DECL PDAT PPDAT515={VEL 100.0,ACC 100.0,APO_DIST 100.0}
DECL E6POS XP770={x 834.883606,y -646.192993,z 1419.58496,a -154.975098,b 4.24509811,c -178.286499,s 2,t 10,e1 0.0,e2 0.0,e3 0.0,e4 0.0,e5 0.0,e6 0.0}
DECL FDAT FP770={TOOL_NO 1,BASE_NO 0,IPO_FRAME #BASE}
DECL PDAT PPDAT516={VEL 100.0,ACC 100.0,APO_DIST 100.0}
DECL E6POS XP771={x 884.407715,y -646.247375,z 1213.34998,a -154.963196,b 4.23633385,c -178.281204,s 2,t 10,e1 0.0,e2 0.0,e3 0.0,e4 0.0,e5 0.0,e6 0.0}
DECL FDAT FP771={TOOL_NO 1,BASE_NO 0,IPO_FRAME #BASE}
DECL PDAT PPDAT517={VEL 100.0,ACC 100.0,APO_DIST 100.0}
DECL E6POS XP772={x 884.420776,y -646.274414,z 1177.65503,a -154.965607,b 4.23612499,c -178.276794,s 2,t 10,e1 0.0,e2 0.0,e3 0.0,e4 0.0,e5 0.0,e6 0.0}
DECL FDAT FP772={TOOL_NO 1,BASE_NO 0,IPO_FRAME #BASE}
DECL LDAT LCPDAT225={VEL 2.0,ACC 100.0,APO_DIST 100.0,APO_FAC 50.0}
DECL E6POS XP773={x 956.251587,y -672.142273,z 1177.66296,a -154.965607,b 4.23677397,c -178.275497,s 2,t 10,e1 0.0,e2 0.0,e3 0.0,e4 0.0,e5 0.0,e6 0.0}
DECL FDAT FP773={TOOL_NO 1,BASE_NO 0,IPO_FRAME #BASE}
DECL LDAT LCPDAT226={VEL 2.0,ACC 100.0,APO_DIST 100.0,APO_FAC 50.0}
DECL E6POS XP774={x 956.253784,y -672.147217,z 1253.29004,a -154.965393,b 4.2372551,c -178.274506,s 2,t 10,e1 0.0,e2 0.0,e3 0.0,e4 0.0,e5 0.0,e6 0.0}
DECL FDAT FP774={TOOL_NO 1,BASE_NO 0,IPO_FRAME #BASE}
DECL LDAT LCPDAT227={VEL 2.0,ACC 100.0,APO_DIST 100.0,APO_FAC 50.0}
DECL E6POS XP775={x 956.25708,y -672.15332,z 1341.07397,a -154.9655,b 4.2373929,c -178.274094,s 2,t 10,e1 0.0,e2 0.0,e3 0.0,e4 0.0,e5 0.0,e6 0.0}
DECL FDAT FP775={TOOL_NO 1,BASE_NO 0,IPO_FRAME #BASE}
DECL PDAT PPDAT518={VEL 100.0,ACC 100.0,APO_DIST 100.0}
DECL E6POS XP776={x 956.26123,y 621.372192,z 1488.15198,a -155.259399,b 5.91821718,c 178.473007,s 2,t 43,e1 0.0,e2 0.0,e3 0.0,e4 0.0,e5 0.0,e6 0.0}
DECL FDAT FP776={TOOL_NO 1,BASE_NO 0,IPO_FRAME #BASE}
DECL PDAT PPDAT519={VEL 100.0,ACC 100.0,APO_DIST 100.0}
DECL E6POS XP777={x 951.221008,y 1494.92102,z 1417.13904,a 164.741592,b -1.48251903,c 173.650696,s 2,t 43,e1 0.0,e2 0.0,e3 0.0,e4 0.0,e5 0.0,e6 0.0}
DECL FDAT FP777={TOOL_NO 1,BASE_NO 0,IPO_FRAME #BASE}
DECL PDAT PPDAT520={VEL 100.0,ACC 100.0,APO_DIST 100.0}
DECL E6POS XP778={x 951.218811,y 1494.91003,z 1304.31799,a 164.741501,b -1.48264694,c 173.651398,s 2,t 43,e1 0.0,e2 0.0,e3 0.0,e4 0.0,e5 0.0,e6 0.0}
DECL FDAT FP778={TOOL_NO 1,BASE_NO 0,IPO_FRAME #BASE}
DECL LDAT LCPDAT228={VEL 2.0,ACC 100.0,APO_DIST 100.0,APO_FAC 50.0}
DECL E6POS XP779={x 951.21698,y 1494.91504,z 1203.42395,a 164.741592,b -1.48277903,c 173.651398,s 2,t 43,e1 0.0,e2 0.0,e3 0.0,e4 0.0,e5 0.0,e6 0.0}
DECL FDAT FP779={TOOL_NO 1,BASE_NO 0,IPO_FRAME #BASE}
DECL LDAT LCPDAT229={VEL 2.0,ACC 100.0,APO_DIST 100.0,APO_FAC 50.0}
DECL E6POS XP780={x 781.836426,y 1615.77795,z 1203.41504,a 164.741699,b -1.48282301,c 173.651199,s 2,t 43,e1 0.0,e2 0.0,e3 0.0,e4 0.0,e5 0.0,e6 0.0}
DECL FDAT FP780={TOOL_NO 1,BASE_NO 0,IPO_FRAME #BASE}
DECL LDAT LCPDAT230={VEL 2.0,ACC 100.0,APO_DIST 100.0,APO_FAC 50.0}
DECL E6POS XP781={x 781.839783,y 1615.78406,z 1295.63196,a 164.741196,b -1.48269701,c 173.650696,s 2,t 43,e1 0.0,e2 0.0,e3 0.0,e4 0.0,e5 0.0,e6 0.0}
DECL FDAT FP781={TOOL_NO 1,BASE_NO 0,IPO_FRAME #BASE}
DECL PDAT PPDAT521={VEL 100.0,ACC 100.0,APO_DIST 100.0}
DECL E6POS XP782={x 781.841492,y 1615.78699,z 1625.56396,a 164.740997,b -1.48261797,c 173.650497,s 2,t 43,e1 0.0,e2 0.0,e3 0.0,e4 0.0,e5 0.0,e6 0.0}
DECL FDAT FP782={TOOL_NO 1,BASE_NO 0,IPO_FRAME #BASE}
DECL PDAT PPDAT522={VEL 100.0,ACC 100.0,APO_DIST 100.0}
DECL E6POS XP783={x 781.886414,y 50.4748688,z 1625.57104,a -152.987396,b 4.59010792,c 178.606796,s 2,t 11,e1 0.0,e2 0.0,e3 0.0,e4 0.0,e5 0.0,e6 0.0}
DECL FDAT FP783={TOOL_NO 1,BASE_NO 0,IPO_FRAME #BASE}
DECL PDAT PPDAT523={VEL 100.0,ACC 100.0,APO_DIST 100.0}
DECL E6POS XP784={x 1625.51196,y 50.4724808,z 1091.81201,a -152.987701,b 4.59131098,c 178.607605,s 2,t 11,e1 0.0,e2 0.0,e3 0.0,e4 0.0,e5 0.0,e6 0.0}
DECL FDAT FP784={TOOL_NO 1,BASE_NO 0,IPO_FRAME #BASE}
DECL PDAT PPDAT524={VEL 100.0,ACC 100.0,APO_DIST 100.0}
DECL E6POS XP785={x 1936.96106,y 50.3517113,z 1091.52197,a 169.965393,b 30.0970707,c 148.691498,s 2,t 10,e1 0.0,e2 0.0,e3 0.0,e4 0.0,e5 0.0,e6 0.0}
DECL FDAT FP785={TOOL_NO 1,BASE_NO 0,IPO_FRAME #BASE}
DECL PDAT PPDAT525={VEL 100.0,ACC 100.0,APO_DIST 100.0}
DECL E6POS XP786={x 2177.73804,y -308.035889,z 1091.83203,a 91.7171021,b 5.48031807,c 146.144806,s 2,t 42,e1 0.0,e2 0.0,e3 0.0,e4 0.0,e5 0.0,e6 0.0}
DECL FDAT FP786={TOOL_NO 1,BASE_NO 0,IPO_FRAME #BASE}
DECL PDAT PPDAT526={VEL 100.0,ACC 100.0,APO_DIST 100.0}
DECL E6POS XP787={x 1894.03699,y -621.732422,z 1187.06897,a 25.7903595,b -5.24155807,c 179.080307,s 2,t 42,e1 0.0,e2 0.0,e3 0.0,e4 0.0,e5 0.0,e6 0.0}
DECL FDAT FP787={TOOL_NO 1,BASE_NO 0,IPO_FRAME #BASE}
DECL PDAT PPDAT527={VEL 100.0,ACC 100.0,APO_DIST 100.0}
DECL E6POS XP788={x 1882.03296,y -621.668518,z 1187.04199,a 25.7881699,b -5.23810196,c 179.0793,s 2,t 42,e1 0.0,e2 0.0,e3 0.0,e4 0.0,e5 0.0,e6 0.0}
DECL FDAT FP788={TOOL_NO 1,BASE_NO 0,IPO_FRAME #BASE}
DECL LDAT LCPDAT231={VEL 2.0,ACC 100.0,APO_DIST 100.0,APO_FAC 50.0}
DECL E6POS XP789={x 1807.823,y -621.600098,z 1187.02002,a 25.1856403,b -5.23544598,c 179.079895,s 2,t 42,e1 0.0,e2 0.0,e3 0.0,e4 0.0,e5 0.0,e6 0.0}
DECL FDAT FP789={TOOL_NO 1,BASE_NO 0,IPO_FRAME #BASE}
DECL LDAT LCPDAT232={VEL 2.0,ACC 100.0,APO_DIST 100.0,APO_FAC 50.0}
DECL E6POS XP790={x 1807.828,y -621.599976,z 1272.56396,a 25.1849709,b -5.2358942,c 179.080093,s 2,t 42,e1 0.0,e2 0.0,e3 0.0,e4 0.0,e5 0.0,e6 0.0}
DECL FDAT FP790={TOOL_NO 1,BASE_NO 0,IPO_FRAME #BASE}
DECL LDAT LCPDAT233={VEL 2.0,ACC 100.0,APO_DIST 100.0,APO_FAC 50.0}
DECL E6POS XP791={x 1807.82104,y -621.602295,z 1311.28894,a 25.1842403,b -5.23504496,c 179.080795,s 2,t 42,e1 0.0,e2 0.0,e3 0.0,e4 0.0,e5 0.0,e6 0.0}
DECL FDAT FP791={TOOL_NO 1,BASE_NO 0,IPO_FRAME #BASE}
DECL PDAT PPDAT528={VEL 100.0,ACC 100.0,APO_DIST 100.0}
DECL E6POS XP792={x 1807.82495,y 498.553192,z 1311.28796,a 25.1833591,b -5.23463488,c 179.080795,s 2,t 35,e1 0.0,e2 0.0,e3 0.0,e4 0.0,e5 0.0,e6 0.0}
DECL FDAT FP792={TOOL_NO 1,BASE_NO 0,IPO_FRAME #BASE}
DECL PDAT PPDAT529={VEL 100.0,ACC 100.0,APO_DIST 100.0}
DECL E6POS XP793={x 1629.39404,y 957.296875,z 1392.64502,a -14.3889599,b -2.57446599,c -174.841293,s 2,t 43,e1 0.0,e2 0.0,e3 0.0,e4 0.0,e5 0.0,e6 0.0}
DECL FDAT FP793={TOOL_NO 1,BASE_NO 0,IPO_FRAME #BASE}
DECL PDAT PPDAT530={VEL 100.0,ACC 100.0,APO_DIST 100.0}
DECL E6POS XP794={x 1629.39099,y 957.29303,z 1270.86804,a -14.3891497,b -2.57352996,c -174.841599,s 2,t 43,e1 0.0,e2 0.0,e3 0.0,e4 0.0,e5 0.0,e6 0.0}
DECL FDAT FP794={TOOL_NO 1,BASE_NO 0,IPO_FRAME #BASE}
DECL PDAT PPDAT531={VEL 100.0,ACC 100.0,APO_DIST 100.0}
DECL E6POS XP795={x 1629.39795,y 957.297913,z 1263.79199,a -14.3884897,b -2.57415891,c -174.840897,s 2,t 43,e1 0.0,e2 0.0,e3 0.0,e4 0.0,e5 0.0,e6 0.0}
DECL FDAT FP795={TOOL_NO 1,BASE_NO 0,IPO_FRAME #BASE}
DECL LDAT LCPDAT234={VEL 2.0,ACC 100.0,APO_DIST 100.0,APO_FAC 50.0}
DECL E6POS XP796={x 1629.39294,y 957.290588,z 1205.66602,a -14.3889904,b -2.573524,c -174.841293,s 2,t 43,e1 0.0,e2 0.0,e3 0.0,e4 0.0,e5 0.0,e6 0.0}
DECL FDAT FP796={TOOL_NO 1,BASE_NO 0,IPO_FRAME #BASE}
DECL LDAT LCPDAT235={VEL 2.0,ACC 100.0,APO_DIST 100.0,APO_FAC 50.0}
DECL E6POS XP797={x 1751.35901,y 834.430481,z 1205.68005,a -14.3898897,b -2.57414389,c -174.840302,s 2,t 43,e1 0.0,e2 0.0,e3 0.0,e4 0.0,e5 0.0,e6 0.0}
DECL FDAT FP797={TOOL_NO 1,BASE_NO 0,IPO_FRAME #BASE}
DECL LDAT LCPDAT236={VEL 2.0,ACC 100.0,APO_DIST 100.0,APO_FAC 50.0}
DECL E6POS XP798={x 1751.36096,y 834.434082,z 1290.125,a -14.39009,b -2.57477689,c -174.840103,s 2,t 43,e1 0.0,e2 0.0,e3 0.0,e4 0.0,e5 0.0,e6 0.0}
DECL FDAT FP798={TOOL_NO 1,BASE_NO 0,IPO_FRAME #BASE}
DECL PDAT PPDAT532={VEL 100.0,ACC 100.0,APO_DIST 100.0}
DECL E6POS XP799={x 1482.72302,y 101.339798,z 1842.39502,a -14.3908005,b -2.57482505,c -174.840393,s 2,t 43,e1 0.0,e2 0.0,e3 0.0,e4 0.0,e5 0.0,e6 0.0}
DECL FDAT FP799={TOOL_NO 1,BASE_NO 0,IPO_FRAME #BASE}
DECL PDAT PPDAT533={VEL 100.0,ACC 100.0,APO_DIST 100.0}
DECL E6POS XP800={x 1967.19495,y -1208.297,z 1007.40997,a 30.6325607,b -2.68640089,c 176.940903,s 2,t 42,e1 0.0,e2 0.0,e3 0.0,e4 0.0,e5 0.0,e6 0.0}
DECL FDAT FP800={TOOL_NO 1,BASE_NO 0,IPO_FRAME #BASE}
DECL PDAT PPDAT534={VEL 100.0,ACC 100.0,APO_DIST 100.0}
DECL E6POS XP801={x 1867.01794,y -1528.33398,z 676.013306,a 26.0535393,b -2.69201303,c 176.927597,s 2,t 42,e1 0.0,e2 0.0,e3 0.0,e4 0.0,e5 0.0,e6 0.0}
DECL FDAT FP801={TOOL_NO 1,BASE_NO 0,IPO_FRAME #BASE}
DECL PDAT PPDAT535={VEL 100.0,ACC 100.0,APO_DIST 100.0}
DECL E6POS XP802={x 1867.14905,y -1528.302,z 632.177185,a 26.0634403,b -2.69869804,c 176.917206,s 2,t 42,e1 0.0,e2 0.0,e3 0.0,e4 0.0,e5 0.0,e6 0.0}
DECL FDAT FP802={TOOL_NO 1,BASE_NO 0,IPO_FRAME #BASE}
DECL LDAT LCPDAT237={VEL 2.0,ACC 100.0,APO_DIST 100.0,APO_FAC 50.0}
DECL E6POS XP803={x 1803.28406,y -1528.18005,z 632.140503,a 26.0650692,b -2.69497204,c 176.921204,s 2,t 42,e1 0.0,e2 0.0,e3 0.0,e4 0.0,e5 0.0,e6 0.0}
DECL FDAT FP803={TOOL_NO 1,BASE_NO 0,IPO_FRAME #BASE}
DECL LDAT LCPDAT238={VEL 2.0,ACC 100.0,APO_DIST 100.0,APO_FAC 50.0}
DECL E6POS XP804={x 1803.28699,y -1528.19104,z 666.373779,a 26.0654392,b -2.69498992,c 176.920303,s 2,t 42,e1 0.0,e2 0.0,e3 0.0,e4 0.0,e5 0.0,e6 0.0}
DECL FDAT FP804={TOOL_NO 1,BASE_NO 0,IPO_FRAME #BASE}
DECL LDAT LCPDAT239={VEL 2.0,ACC 100.0,APO_DIST 100.0,APO_FAC 50.0}
DECL E6POS XP805={x 1803.29004,y -1528.18799,z 707.782471,a 26.0653191,b -2.69489288,c 176.920105,s 2,t 42,e1 0.0,e2 0.0,e3 0.0,e4 0.0,e5 0.0,e6 0.0}
DECL FDAT FP805={TOOL_NO 1,BASE_NO 0,IPO_FRAME #BASE}
DECL PDAT PPDAT536={VEL 100.0,ACC 100.0,APO_DIST 100.0}
DECL E6POS XP806={x 1849.71899,y 504.765503,z 982.790527,a 25.7066708,b -3.66189194,c -178.073196,s 2,t 43,e1 0.0,e2 0.0,e3 0.0,e4 0.0,e5 0.0,e6 0.0}
DECL FDAT FP806={TOOL_NO 1,BASE_NO 0,IPO_FRAME #BASE}
DECL PDAT PPDAT537={VEL 100.0,ACC 100.0,APO_DIST 100.0}
DECL E6POS XP807={x 1526.51599,y 887.347717,z 1356.229,a 119.449997,b -0.79832828,c 176.833496,s 2,t 43,e1 0.0,e2 0.0,e3 0.0,e4 0.0,e5 0.0,e6 0.0}
DECL FDAT FP807={TOOL_NO 1,BASE_NO 0,IPO_FRAME #BASE}
DECL PDAT PPDAT538={VEL 100.0,ACC 100.0,APO_DIST 100.0}
DECL E6POS XP808={x 1117.29504,y 985.80957,z 1503.50098,a -103.3563,b 6.37956905,c -178.578705,s 2,t 11,e1 0.0,e2 0.0,e3 0.0,e4 0.0,e5 0.0,e6 0.0}
DECL FDAT FP808={TOOL_NO 1,BASE_NO 0,IPO_FRAME #BASE}
DECL PDAT PPDAT539={VEL 100.0,ACC 100.0,APO_DIST 100.0}
DECL E6POS XP809={x 1110.35498,y 986.373596,z 1199.61401,a -104.191902,b 6.3782239,c -178.580399,s 2,t 11,e1 0.0,e2 0.0,e3 0.0,e4 0.0,e5 0.0,e6 0.0}
DECL FDAT FP809={TOOL_NO 1,BASE_NO 0,IPO_FRAME #BASE}
DECL LDAT LCPDAT240={VEL 2.0,ACC 100.0,APO_DIST 100.0,APO_FAC 50.0}
DECL E6POS XP810={x 1110.35706,y 986.37439,z 1177.31006,a -104.191597,b 6.37824202,c -178.580093,s 2,t 11,e1 0.0,e2 0.0,e3 0.0,e4 0.0,e5 0.0,e6 0.0}
DECL FDAT FP810={TOOL_NO 1,BASE_NO 0,IPO_FRAME #BASE}
DECL LDAT LCPDAT241={VEL 2.0,ACC 100.0,APO_DIST 100.0,APO_FAC 50.0}
DECL E6POS XP811={x 1060.698,y 922.256287,z 1177.30701,a -104.191704,b 6.3783679,c -178.580093,s 2,t 11,e1 0.0,e2 0.0,e3 0.0,e4 0.0,e5 0.0,e6 0.0}
DECL FDAT FP811={TOOL_NO 1,BASE_NO 0,IPO_FRAME #BASE}
DECL LDAT LCPDAT242={VEL 2.0,ACC 100.0,APO_DIST 100.0,APO_FAC 50.0}
DECL E6POS XP812={x 1060.70605,y 922.260193,z 1248.45898,a -104.1922,b 6.37897682,c -178.580002,s 2,t 11,e1 0.0,e2 0.0,e3 0.0,e4 0.0,e5 0.0,e6 0.0}
DECL FDAT FP812={TOOL_NO 1,BASE_NO 0,IPO_FRAME #BASE}
DECL LDAT LCPDAT243={VEL 2.0,ACC 100.0,APO_DIST 100.0,APO_FAC 50.0}
DECL E6POS XP813={x 1060.70801,y 922.260986,z 1325.92102,a -104.193199,b 6.37862921,c -178.5802,s 2,t 11,e1 0.0,e2 0.0,e3 0.0,e4 0.0,e5 0.0,e6 0.0}
DECL FDAT FP813={TOOL_NO 1,BASE_NO 0,IPO_FRAME #BASE}
DECL PDAT PPDAT540={VEL 100.0,ACC 100.0,APO_DIST 100.0}
DECL E6POS XP814={x 1007.14001,y -531.034973,z 1325.93103,a -154.515793,b 6.37904882,c -178.579803,s 2,t 10,e1 0.0,e2 0.0,e3 0.0,e4 0.0,e5 0.0,e6 0.0}
DECL FDAT FP814={TOOL_NO 1,BASE_NO 0,IPO_FRAME #BASE}
DECL PDAT PPDAT541={VEL 100.0,ACC 100.0,APO_DIST 100.0}
DECL E6POS XP815={x 662.151917,y -1577.61401,z 1042.82104,a -155.219803,b 2.91244411,c -175.284103,s 2,t 10,e1 0.0,e2 0.0,e3 0.0,e4 0.0,e5 0.0,e6 0.0}
DECL FDAT FP815={TOOL_NO 1,BASE_NO 0,IPO_FRAME #BASE}
DECL PDAT PPDAT542={VEL 100.0,ACC 100.0,APO_DIST 100.0}
DECL E6POS XP816={x 595.804382,y -1577.60999,z 610.217285,a -155.219498,b 2.91238999,c -175.284607,s 2,t 10,e1 0.0,e2 0.0,e3 0.0,e4 0.0,e5 0.0,e6 0.0}
DECL FDAT FP816={TOOL_NO 1,BASE_NO 0,IPO_FRAME #BASE}
DECL PDAT PPDAT543={VEL 100.0,ACC 100.0,APO_DIST 100.0}
DECL E6POS XP817={x 677.520874,y -1577.67395,z 616.163086,a -155.236404,b 0.510486484,c -174.949493,s 2,t 10,e1 0.0,e2 0.0,e3 0.0,e4 0.0,e5 0.0,e6 0.0}
DECL FDAT FP817={TOOL_NO 1,BASE_NO 0,IPO_FRAME #BASE}
DECL PDAT PPDAT544={VEL 100.0,ACC 100.0,APO_DIST 100.0}
DECL E6POS XP818={x 680.30188,y -1577.672,z 616.161621,a -155.236694,b 0.510483205,c -174.949905,s 2,t 10,e1 0.0,e2 0.0,e3 0.0,e4 0.0,e5 0.0,e6 0.0}
DECL FDAT FP818={TOOL_NO 1,BASE_NO 0,IPO_FRAME #BASE}
DECL LDAT LCPDAT244={VEL 2.0,ACC 100.0,APO_DIST 100.0,APO_FAC 50.0}
DECL E6POS XP819={x 729.268921,y -1577.66602,z 614.958984,a -155.235901,b 0.510274529,c -174.950394,s 2,t 10,e1 0.0,e2 0.0,e3 0.0,e4 0.0,e5 0.0,e6 0.0}
DECL FDAT FP819={TOOL_NO 1,BASE_NO 0,IPO_FRAME #BASE}
DECL LDAT LCPDAT245={VEL 2.0,ACC 100.0,APO_DIST 100.0,APO_FAC 50.0}
DECL E6POS XP820={x 729.266174,y -1577.66895,z 665.128723,a -155.235794,b 0.510224879,c -174.950699,s 2,t 10,e1 0.0,e2 0.0,e3 0.0,e4 0.0,e5 0.0,e6 0.0}
DECL FDAT FP820={TOOL_NO 1,BASE_NO 0,IPO_FRAME #BASE}
DECL LDAT LCPDAT246={VEL 2.0,ACC 100.0,APO_DIST 100.0,APO_FAC 50.0}
DECL E6POS XP821={x 729.262085,y -1577.66003,z 715.29657,a -155.235703,b 0.510212183,c -174.951202,s 2,t 10,e1 0.0,e2 0.0,e3 0.0,e4 0.0,e5 0.0,e6 0.0}
DECL FDAT FP821={TOOL_NO 1,BASE_NO 0,IPO_FRAME #BASE}
DECL PDAT PPDAT545={VEL 100.0,ACC 100.0,APO_DIST 100.0}
DECL E6POS XP822={x 1350.92798,y -438.835693,z 1277.92603,a -155.235504,b 0.510017395,c -174.951096,s 2,t 2,e1 0.0,e2 0.0,e3 0.0,e4 0.0,e5 0.0,e6 0.0}
DECL FDAT FP822={TOOL_NO 1,BASE_NO 0,IPO_FRAME #BASE}
DECL PDAT PPDAT546={VEL 100.0,ACC 100.0,APO_DIST 100.0}
DECL E6POS XP823={x 1350.94495,y -65.3104172,z 1277.97803,a -155.459106,b 3.8784039,c -179.287598,s 2,t 10,e1 0.0,e2 0.0,e3 0.0,e4 0.0,e5 0.0,e6 0.0}
DECL FDAT FP823={TOOL_NO 1,BASE_NO 0,IPO_FRAME #BASE}
DECL PDAT PPDAT547={VEL 100.0,ACC 100.0,APO_DIST 100.0}
DECL E6POS XP824={x 1350.95801,y 508.329315,z 1277.97095,a -103.423302,b 3.87848401,c -179.288406,s 2,t 11,e1 0.0,e2 0.0,e3 0.0,e4 0.0,e5 0.0,e6 0.0}
DECL FDAT FP824={TOOL_NO 1,BASE_NO 0,IPO_FRAME #BASE}
DECL PDAT PPDAT548={VEL 100.0,ACC 100.0,APO_DIST 100.0}
DECL E6POS XP825={x 976.178101,y 799.219421,z 1277.97095,a -103.422897,b 3.87840891,c -179.288498,s 2,t 11,e1 0.0,e2 0.0,e3 0.0,e4 0.0,e5 0.0,e6 0.0}
DECL FDAT FP825={TOOL_NO 1,BASE_NO 0,IPO_FRAME #BASE}
DECL PDAT PPDAT549={VEL 100.0,ACC 100.0,APO_DIST 100.0}
DECL E6POS XP826={x 976.189697,y 799.22113,z 1265.927,a -103.4245,b 3.87825489,c -179.287796,s 2,t 11,e1 0.0,e2 0.0,e3 0.0,e4 0.0,e5 0.0,e6 0.0}
DECL FDAT FP826={TOOL_NO 1,BASE_NO 0,IPO_FRAME #BASE}
DECL LDAT LCPDAT247={VEL 2.0,ACC 100.0,APO_DIST 100.0,APO_FAC 50.0}
DECL E6POS XP827={x 973.25177,y 802.428528,z 1180.17896,a -104.262299,b 3.87858891,c -179.288193,s 2,t 11,e1 0.0,e2 0.0,e3 0.0,e4 0.0,e5 0.0,e6 0.0}
DECL FDAT FP827={TOOL_NO 1,BASE_NO 0,IPO_FRAME #BASE}
DECL LDAT LCPDAT248={VEL 2.0,ACC 100.0,APO_DIST 100.0,APO_FAC 50.0}
DECL E6POS XP828={x 903.986694,y 734.74292,z 1180.17896,a -104.262199,b 3.87883902,c -179.288101,s 2,t 11,e1 0.0,e2 0.0,e3 0.0,e4 0.0,e5 0.0,e6 0.0}
DECL FDAT FP828={TOOL_NO 1,BASE_NO 0,IPO_FRAME #BASE}
DECL LDAT LCPDAT249={VEL 2.0,ACC 100.0,APO_DIST 100.0,APO_FAC 50.0}
DECL E6POS XP829={x 903.989075,y 691.025574,z 1431.854,a -104.2621,b 3.87912607,c -179.287994,s 2,t 11,e1 0.0,e2 0.0,e3 0.0,e4 0.0,e5 0.0,e6 0.0}
DECL FDAT FP829={TOOL_NO 1,BASE_NO 0,IPO_FRAME #BASE}
DECL PDAT PPDAT550={VEL 100.0,ACC 100.0,APO_DIST 100.0}
DECL E6POS XP830={x 1242.453,y 383.157196,z 1431.854,a -65.0922165,b 1.82727897,c -174.843307,s 2,t 11,e1 0.0,e2 0.0,e3 0.0,e4 0.0,e5 0.0,e6 0.0}
DECL FDAT FP830={TOOL_NO 1,BASE_NO 0,IPO_FRAME #BASE}
DECL PDAT PPDAT551={VEL 100.0,ACC 100.0,APO_DIST 100.0}
DECL E6POS XP831={x 1242.526,y -1715.71497,z 1090.12195,a -65.0943909,b 1.824404,c -174.841507,s 2,t 10,e1 0.0,e2 0.0,e3 0.0,e4 0.0,e5 0.0,e6 0.0}
DECL FDAT FP831={TOOL_NO 1,BASE_NO 0,IPO_FRAME #BASE}
DECL PDAT PPDAT552={VEL 100.0,ACC 100.0,APO_DIST 100.0}
DECL E6POS XP832={x 1267.51099,y -2121.16797,z 696.45282,a -64.79319,b -2.43663502,c -176.824097,s 2,t 10,e1 0.0,e2 0.0,e3 0.0,e4 0.0,e5 0.0,e6 0.0}
DECL FDAT FP832={TOOL_NO 1,BASE_NO 0,IPO_FRAME #BASE}
DECL PDAT PPDAT553={VEL 100.0,ACC 100.0,APO_DIST 100.0}
DECL E6POS XP833={x 1268.06104,y -2138.6001,z 629.002625,a -64.8109665,b -2.74127197,c -176.339798,s 2,t 10,e1 0.0,e2 0.0,e3 0.0,e4 0.0,e5 0.0,e6 0.0}
DECL FDAT FP833={TOOL_NO 1,BASE_NO 0,IPO_FRAME #BASE}
DECL LDAT LCPDAT250={VEL 2.0,ACC 100.0,APO_DIST 100.0,APO_FAC 50.0}
DECL E6POS XP834={x 1267.37195,y -2113.87012,z 626.005981,a -64.8136368,b -2.71599889,c -176.349594,s 2,t 10,e1 0.0,e2 0.0,e3 0.0,e4 0.0,e5 0.0,e6 0.0}
DECL FDAT FP834={TOOL_NO 1,BASE_NO 0,IPO_FRAME #BASE}
DECL LDAT LCPDAT251={VEL 2.0,ACC 100.0,APO_DIST 100.0,APO_FAC 50.0}
DECL E6POS XP835={x 1267.10999,y -2080.51807,z 625.848328,a -64.8051834,b -2.70687294,c -176.356506,s 2,t 10,e1 0.0,e2 0.0,e3 0.0,e4 0.0,e5 0.0,e6 0.0}
DECL FDAT FP835={TOOL_NO 1,BASE_NO 0,IPO_FRAME #BASE}
DECL LDAT LCPDAT252={VEL 2.0,ACC 100.0,APO_DIST 100.0,APO_FAC 50.0}
DECL E6POS XP836={x 1267.10901,y -2080.51611,z 624.96228,a -64.8052521,b -2.70639491,c -176.356598,s 2,t 10,e1 0.0,e2 0.0,e3 0.0,e4 0.0,e5 0.0,e6 0.0}
DECL FDAT FP836={TOOL_NO 1,BASE_NO 0,IPO_FRAME #BASE}
DECL LDAT LCPDAT253={VEL 2.0,ACC 100.0,APO_DIST 100.0,APO_FAC 50.0}
DECL E6POS XP837={x 1284.23096,y -2080.74902,z 625.221313,a -64.8089066,b -2.72878504,c -176.344299,s 2,t 10,e1 0.0,e2 0.0,e3 0.0,e4 0.0,e5 0.0,e6 0.0}
DECL FDAT FP837={TOOL_NO 1,BASE_NO 0,IPO_FRAME #BASE}
DECL LDAT LCPDAT254={VEL 2.0,ACC 100.0,APO_DIST 100.0,APO_FAC 50.0}
DECL E6POS XP838={x 1284.21899,y -2080.75,z 674.30957,a -64.8095093,b -2.728158,c -176.344498,s 2,t 10,e1 0.0,e2 0.0,e3 0.0,e4 0.0,e5 0.0,e6 0.0}
DECL FDAT FP838={TOOL_NO 1,BASE_NO 0,IPO_FRAME #BASE}
DECL LDAT LCPDAT255={VEL 2.0,ACC 100.0,APO_DIST 100.0,APO_FAC 50.0}
DECL E6POS XP839={x 1284.21301,y -2080.75098,z 781.889709,a -64.8102188,b -2.72803593,c -176.344498,s 2,t 10,e1 0.0,e2 0.0,e3 0.0,e4 0.0,e5 0.0,e6 0.0}
DECL FDAT FP839={TOOL_NO 1,BASE_NO 0,IPO_FRAME #BASE}
DECL PDAT PPDAT554={VEL 100.0,ACC 100.0,APO_DIST 100.0}
DECL E6POS XP840={x 1284.33301,y 158.871704,z 1306.61304,a -64.8253937,b 1.14583802,c -174.523804,s 2,t 11,e1 0.0,e2 0.0,e3 0.0,e4 0.0,e5 0.0,e6 0.0}
DECL FDAT FP840={TOOL_NO 1,BASE_NO 0,IPO_FRAME #BASE}
DECL PDAT PPDAT555={VEL 100.0,ACC 100.0,APO_DIST 100.0}
DECL E6POS XP841={x 1590.53296,y 626.546387,z 1306.651,a -14.1000004,b -1.28675902,c -174.4617,s 2,t 11,e1 0.0,e2 0.0,e3 0.0,e4 0.0,e5 0.0,e6 0.0}
DECL FDAT FP841={TOOL_NO 1,BASE_NO 0,IPO_FRAME #BASE}
DECL PDAT PPDAT556={VEL 100.0,ACC 100.0,APO_DIST 100.0}
DECL E6POS XP842={x 1716.79199,y 897.809082,z 1262.11096,a -13.9702301,b -1.29123998,c -174.459503,s 2,t 11,e1 0.0,e2 0.0,e3 0.0,e4 0.0,e5 0.0,e6 0.0}
DECL FDAT FP842={TOOL_NO 1,BASE_NO 0,IPO_FRAME #BASE}
DECL PDAT PPDAT557={VEL 100.0,ACC 100.0,APO_DIST 100.0}
DECL E6POS XP843={x 1716.79199,y 897.806274,z 1247.396,a -13.9698601,b -1.29120898,c -174.459,s 2,t 11,e1 0.0,e2 0.0,e3 0.0,e4 0.0,e5 0.0,e6 0.0}
DECL FDAT FP843={TOOL_NO 1,BASE_NO 0,IPO_FRAME #BASE}
DECL LDAT LCPDAT256={VEL 2.0,ACC 100.0,APO_DIST 100.0,APO_FAC 50.0}
DECL E6POS XP844={x 1716.78198,y 897.80249,z 1198.69897,a -13.9701004,b -1.29035699,c -174.459396,s 2,t 11,e1 0.0,e2 0.0,e3 0.0,e4 0.0,e5 0.0,e6 0.0}
DECL FDAT FP844={TOOL_NO 1,BASE_NO 0,IPO_FRAME #BASE}
DECL LDAT LCPDAT257={VEL 2.0,ACC 100.0,APO_DIST 100.0,APO_FAC 50.0}
DECL E6POS XP845={x 1802.52795,y 828.709717,z 1198.69604,a -13.9702501,b -1.29001105,c -174.459305,s 2,t 11,e1 0.0,e2 0.0,e3 0.0,e4 0.0,e5 0.0,e6 0.0}
DECL FDAT FP845={TOOL_NO 1,BASE_NO 0,IPO_FRAME #BASE}
DECL LDAT LCPDAT258={VEL 2.0,ACC 100.0,APO_DIST 100.0,APO_FAC 50.0}
DECL E6POS XP846={x 1802.51294,y 761.127502,z 1198.72302,a -13.9681501,b -1.29168904,c -174.458298,s 2,t 11,e1 0.0,e2 0.0,e3 0.0,e4 0.0,e5 0.0,e6 0.0}
DECL FDAT FP846={TOOL_NO 1,BASE_NO 0,IPO_FRAME #BASE}
DECL PDAT PPDAT558={VEL 100.0,ACC 100.0,APO_DIST 100.0}
DECL E6POS XP847={x 1802.50598,y -336.506287,z 1185.67297,a 118.019897,b 4.52842808,c 174.709198,s 2,t 34,e1 0.0,e2 0.0,e3 0.0,e4 0.0,e5 0.0,e6 0.0}
DECL FDAT FP847={TOOL_NO 1,BASE_NO 0,IPO_FRAME #BASE}
DECL PDAT PPDAT559={VEL 100.0,ACC 100.0,APO_DIST 100.0}
DECL E6POS XP848={x 1270.18604,y -947.062622,z 660.983521,a 112.980698,b 4.33244419,c 178.080505,s 2,t 34,e1 0.0,e2 0.0,e3 0.0,e4 0.0,e5 0.0,e6 0.0}
DECL FDAT FP848={TOOL_NO 1,BASE_NO 0,IPO_FRAME #BASE}
DECL PDAT PPDAT560={VEL 100.0,ACC 100.0,APO_DIST 100.0}
DECL E6POS XP849={x 1286.21497,y -986.133179,z 597.794983,a 112.979897,b 4.33160305,c 178.080902,s 2,t 34,e1 0.0,e2 0.0,e3 0.0,e4 0.0,e5 0.0,e6 0.0}
DECL FDAT FP849={TOOL_NO 1,BASE_NO 0,IPO_FRAME #BASE}
DECL LDAT LCPDAT259={VEL 2.0,ACC 100.0,APO_DIST 100.0,APO_FAC 50.0}
DECL E6POS XP850={x 1286.00305,y -1018.45898,z 597.88147,a 113.2043,b 4.06272316,c 178.724106,s 2,t 34,e1 0.0,e2 0.0,e3 0.0,e4 0.0,e5 0.0,e6 0.0}
DECL FDAT FP850={TOOL_NO 1,BASE_NO 0,IPO_FRAME #BASE}
DECL LDAT LCPDAT260={VEL 2.0,ACC 100.0,APO_DIST 100.0,APO_FAC 50.0}
DECL E6POS XP851={x 1274.45605,y -1018.44501,z 598.83728,a 113.204597,b 4.06176376,c 178.724594,s 2,t 34,e1 0.0,e2 0.0,e3 0.0,e4 0.0,e5 0.0,e6 0.0}
DECL FDAT FP851={TOOL_NO 1,BASE_NO 0,IPO_FRAME #BASE}
DECL LDAT LCPDAT261={VEL 2.0,ACC 100.0,APO_DIST 100.0,APO_FAC 50.0}
DECL E6POS XP852={x 1274.45996,y -1018.448,z 627.330078,a 113.205299,b 4.06202507,c 178.724503,s 2,t 34,e1 0.0,e2 0.0,e3 0.0,e4 0.0,e5 0.0,e6 0.0}
DECL FDAT FP852={TOOL_NO 1,BASE_NO 0,IPO_FRAME #BASE}
DECL LDAT LCPDAT262={VEL 2.0,ACC 100.0,APO_DIST 100.0,APO_FAC 50.0}
DECL E6POS XP853={x 1274.47095,y -1018.46503,z 647.700317,a 113.2052,b 4.06336021,c 178.723801,s 2,t 34,e1 0.0,e2 0.0,e3 0.0,e4 0.0,e5 0.0,e6 0.0}
DECL FDAT FP853={TOOL_NO 1,BASE_NO 0,IPO_FRAME #BASE}
DECL PDAT PPDAT561={VEL 100.0,ACC 100.0,APO_DIST 100.0}
DECL E6POS XP854={x 1274.40405,y 438.174194,z 1449.75903,a 113.028397,b 1.96038795,c 176.1409,s 2,t 35,e1 0.0,e2 0.0,e3 0.0,e4 0.0,e5 0.0,e6 0.0}
DECL FDAT FP854={TOOL_NO 1,BASE_NO 0,IPO_FRAME #BASE}
DECL PDAT PPDAT562={VEL 100.0,ACC 100.0,APO_DIST 100.0}
DECL E6POS XP855={x 1274.41199,y 579.304382,z 1449.76697,a -174.676498,b 7.10730505,c 176.619904,s 2,t 43,e1 0.0,e2 0.0,e3 0.0,e4 0.0,e5 0.0,e6 0.0}
DECL FDAT FP855={TOOL_NO 1,BASE_NO 0,IPO_FRAME #BASE}
DECL PDAT PPDAT563={VEL 100.0,ACC 100.0,APO_DIST 100.0}
DECL E6POS XP856={x 1274.41699,y 964.305115,z 1449.76404,a -153.690308,b 6.61543608,c -179.989594,s 2,t 35,e1 0.0,e2 0.0,e3 0.0,e4 0.0,e5 0.0,e6 0.0}
DECL FDAT FP856={TOOL_NO 1,BASE_NO 0,IPO_FRAME #BASE}
DECL PDAT PPDAT564={VEL 100.0,ACC 100.0,APO_DIST 100.0}
DECL E6POS XP857={x 758.336426,y 1284.67102,z 1449.76001,a 165.206497,b 2.00212693,c 176.736298,s 2,t 35,e1 0.0,e2 0.0,e3 0.0,e4 0.0,e5 0.0,e6 0.0}
DECL FDAT FP857={TOOL_NO 1,BASE_NO 0,IPO_FRAME #BASE}
DECL PDAT PPDAT565={VEL 100.0,ACC 100.0,APO_DIST 100.0}
DECL E6POS XP858={x 865.113892,y 1552.07104,z 1237.68701,a 166.427094,b 2.00283194,c 176.733902,s 2,t 35,e1 0.0,e2 0.0,e3 0.0,e4 0.0,e5 0.0,e6 0.0}
DECL FDAT FP858={TOOL_NO 1,BASE_NO 0,IPO_FRAME #BASE}
DECL PDAT PPDAT566={VEL 100.0,ACC 100.0,APO_DIST 100.0}
DECL E6POS XP859={x 865.110718,y 1552.06494,z 1225.62695,a 166.426804,b 2.00282502,c 176.7341,s 2,t 35,e1 0.0,e2 0.0,e3 0.0,e4 0.0,e5 0.0,e6 0.0}
DECL FDAT FP859={TOOL_NO 1,BASE_NO 0,IPO_FRAME #BASE}
DECL LDAT LCPDAT263={VEL 2.0,ACC 100.0,APO_DIST 100.0,APO_FAC 50.0}
DECL E6POS XP860={x 865.113098,y 1552.06201,z 1174.51501,a 166.426193,b 2.00270891,c 176.733994,s 2,t 35,e1 0.0,e2 0.0,e3 0.0,e4 0.0,e5 0.0,e6 0.0}
DECL FDAT FP860={TOOL_NO 1,BASE_NO 0,IPO_FRAME #BASE}
DECL LDAT LCPDAT264={VEL 2.0,ACC 100.0,APO_DIST 100.0,APO_FAC 50.0}
DECL E6POS XP861={x 739.028076,y 1608.69604,z 1174.51501,a 166.426193,b 2.00264096,c 176.733994,s 2,t 35,e1 0.0,e2 0.0,e3 0.0,e4 0.0,e5 0.0,e6 0.0}
DECL FDAT FP861={TOOL_NO 1,BASE_NO 0,IPO_FRAME #BASE}
DECL LDAT LCPDAT265={VEL 2.0,ACC 100.0,APO_DIST 100.0,APO_FAC 50.0}
DECL E6POS XP862={x 739.030212,y 1608.69299,z 1249.495,a 166.425995,b 2.0026021,c 176.733093,s 2,t 35,e1 0.0,e2 0.0,e3 0.0,e4 0.0,e5 0.0,e6 0.0}
DECL FDAT FP862={TOOL_NO 1,BASE_NO 0,IPO_FRAME #BASE}
DECL PDAT PPDAT567={VEL 100.0,ACC 100.0,APO_DIST 100.0}
DECL E6POS XP863={x 977.82428,y 601.907227,z 1521.28406,a -150.784698,b 2.0027411,c 176.732895,s 2,t 11,e1 0.0,e2 0.0,e3 0.0,e4 0.0,e5 0.0,e6 0.0}
DECL FDAT FP863={TOOL_NO 1,BASE_NO 0,IPO_FRAME #BASE}
DECL PDAT PPDAT568={VEL 100.0,ACC 100.0,APO_DIST 100.0}
DECL E6POS XP864={x 977.828918,y -339.057892,z 1521.28296,a -150.784805,b 2.0027051,c 176.733093,s 2,t 10,e1 0.0,e2 0.0,e3 0.0,e4 0.0,e5 0.0,e6 0.0}
DECL FDAT FP864={TOOL_NO 1,BASE_NO 0,IPO_FRAME #BASE}
DECL PDAT PPDAT569={VEL 100.0,ACC 100.0,APO_DIST 100.0}
DECL E6POS XP865={x 667.386719,y -1536.68201,z 1024.74194,a -155.497299,b 5.11866999,c -174.992004,s 2,t 10,e1 0.0,e2 0.0,e3 0.0,e4 0.0,e5 0.0,e6 0.0}
DECL FDAT FP865={TOOL_NO 1,BASE_NO 0,IPO_FRAME #BASE}
DECL PDAT PPDAT570={VEL 100.0,ACC 100.0,APO_DIST 100.0}
DECL E6POS XP866={x 622.895874,y -1574.84204,z 545.977112,a -155.458801,b 2.811517,c -174.407898,s 2,t 10,e1 0.0,e2 0.0,e3 0.0,e4 0.0,e5 0.0,e6 0.0}
DECL FDAT FP866={TOOL_NO 1,BASE_NO 0,IPO_FRAME #BASE}
DECL PDAT PPDAT571={VEL 100.0,ACC 100.0,APO_DIST 100.0}
DECL E6POS XP867={x 672.657288,y -1574.83606,z 545.976685,a -155.459,b 2.81164193,c -174.408707,s 2,t 10,e1 0.0,e2 0.0,e3 0.0,e4 0.0,e5 0.0,e6 0.0}
DECL FDAT FP867={TOOL_NO 1,BASE_NO 0,IPO_FRAME #BASE}
DECL LDAT LCPDAT266={VEL 2.0,ACC 100.0,APO_DIST 100.0,APO_FAC 50.0}
DECL E6POS XP868={x 721.0354,y -1574.83899,z 545.978271,a -155.458801,b 2.8112781,c -174.408005,s 2,t 10,e1 0.0,e2 0.0,e3 0.0,e4 0.0,e5 0.0,e6 0.0}
DECL FDAT FP868={TOOL_NO 1,BASE_NO 0,IPO_FRAME #BASE}
DECL LDAT LCPDAT267={VEL 2.0,ACC 100.0,APO_DIST 100.0,APO_FAC 50.0}
DECL E6POS XP869={x 724.281128,y -1574.85596,z 573.222107,a -155.458694,b 2.81117201,c -174.406998,s 2,t 10,e1 0.0,e2 0.0,e3 0.0,e4 0.0,e5 0.0,e6 0.0}
DECL FDAT FP869={TOOL_NO 1,BASE_NO 0,IPO_FRAME #BASE}
DECL LDAT LCPDAT268={VEL 2.0,ACC 100.0,APO_DIST 100.0,APO_FAC 50.0}
DECL E6POS XP870={x 724.284973,y -1574.86401,z 633.002014,a -155.458694,b 2.81121707,c -174.406693,s 2,t 10,e1 0.0,e2 0.0,e3 0.0,e4 0.0,e5 0.0,e6 0.0}
DECL FDAT FP870={TOOL_NO 1,BASE_NO 0,IPO_FRAME #BASE}
DECL LDAT LCPDAT269={VEL 2.0,ACC 100.0,APO_DIST 100.0,APO_FAC 50.0}
DECL E6POS XP871={x 724.276611,y -1574.85303,z 730.688904,a -155.460098,b 2.81144595,c -174.407898,s 2,t 10,e1 0.0,e2 0.0,e3 0.0,e4 0.0,e5 0.0,e6 0.0}
DECL FDAT FP871={TOOL_NO 1,BASE_NO 0,IPO_FRAME #BASE}
DECL PDAT PPDAT572={VEL 100.0,ACC 100.0,APO_DIST 100.0}
DECL E6POS XP872={x 1196.31104,y -12.7953701,z 1384.39001,a -155.803299,b 5.08000183,c -179.398697,s 2,t 10,e1 0.0,e2 0.0,e3 0.0,e4 0.0,e5 0.0,e6 0.0}
DECL FDAT FP872={TOOL_NO 1,BASE_NO 0,IPO_FRAME #BASE}
DECL PDAT PPDAT573={VEL 100.0,ACC 100.0,APO_DIST 100.0}
DECL E6POS XP873={x 988.161072,y 807.089172,z 1384.35095,a -104.207802,b 7.43646288,c -177.310806,s 2,t 11,e1 0.0,e2 0.0,e3 0.0,e4 0.0,e5 0.0,e6 0.0}
DECL FDAT FP873={TOOL_NO 1,BASE_NO 0,IPO_FRAME #BASE}
DECL PDAT PPDAT574={VEL 100.0,ACC 100.0,APO_DIST 100.0}
DECL E6POS XP874={x 966.663086,y 799.905518,z 1213.52795,a -104.207497,b 7.43645382,c -177.310394,s 2,t 11,e1 0.0,e2 0.0,e3 0.0,e4 0.0,e5 0.0,e6 0.0}
DECL FDAT FP874={TOOL_NO 1,BASE_NO 0,IPO_FRAME #BASE}
DECL PDAT PPDAT575={VEL 100.0,ACC 100.0,APO_DIST 100.0}
DECL E6POS XP875={x 968.942078,y 800.869324,z 1193.94604,a -104.704903,b 7.43691778,c -177.309402,s 2,t 11,e1 0.0,e2 0.0,e3 0.0,e4 0.0,e5 0.0,e6 0.0}
DECL FDAT FP875={TOOL_NO 1,BASE_NO 0,IPO_FRAME #BASE}
DECL LDAT LCPDAT270={VEL 2.0,ACC 100.0,APO_DIST 100.0,APO_FAC 50.0}
DECL E6POS XP876={x 968.950012,y 800.86908,z 1184.78003,a -104.703697,b 7.43699217,c -177.3078,s 2,t 11,e1 0.0,e2 0.0,e3 0.0,e4 0.0,e5 0.0,e6 0.0}
DECL FDAT FP876={TOOL_NO 1,BASE_NO 0,IPO_FRAME #BASE}
DECL LDAT LCPDAT271={VEL 2.0,ACC 100.0,APO_DIST 100.0,APO_FAC 50.0}
DECL E6POS XP877={x 910.592285,y 742.152527,z 1184.78796,a -104.703499,b 7.43762779,c -177.307297,s 2,t 11,e1 0.0,e2 0.0,e3 0.0,e4 0.0,e5 0.0,e6 0.0}
DECL FDAT FP877={TOOL_NO 1,BASE_NO 0,IPO_FRAME #BASE}
DECL LDAT LCPDAT272={VEL 2.0,ACC 100.0,APO_DIST 100.0,APO_FAC 50.0}
DECL E6POS XP878={x 910.58429,y 742.146606,z 1226.82104,a -104.703697,b 7.43728113,c -177.3078,s 2,t 11,e1 0.0,e2 0.0,e3 0.0,e4 0.0,e5 0.0,e6 0.0}
DECL FDAT FP878={TOOL_NO 1,BASE_NO 0,IPO_FRAME #BASE}
DECL PDAT PPDAT576={VEL 100.0,ACC 100.0,APO_DIST 100.0}
DECL E6POS XP879={x 941.989319,y 683.767883,z 1368.15906,a -104.703598,b 7.43723583,c -177.3078,s 2,t 11,e1 0.0,e2 0.0,e3 0.0,e4 0.0,e5 0.0,e6 0.0}
DECL FDAT FP879={TOOL_NO 1,BASE_NO 0,IPO_FRAME #BASE}
DECL PDAT PPDAT577={VEL 100.0,ACC 100.0,APO_DIST 100.0}
DECL E6POS XP880={x 1528.52197,y 420.196503,z 1368.17505,a 25.5136395,b -4.00302076,c -174.884094,s 2,t 43,e1 0.0,e2 0.0,e3 0.0,e4 0.0,e5 0.0,e6 0.0}
DECL FDAT FP880={TOOL_NO 1,BASE_NO 0,IPO_FRAME #BASE}
DECL PDAT PPDAT578={VEL 100.0,ACC 100.0,APO_DIST 100.0}
DECL E6POS XP881={x 1860.85901,y -1558.21399,z 642.981689,a 25.7883205,b -1.25623298,c 176.261795,s 2,t 34,e1 0.0,e2 0.0,e3 0.0,e4 0.0,e5 0.0,e6 0.0}
DECL FDAT FP881={TOOL_NO 1,BASE_NO 0,IPO_FRAME #BASE}
DECL PDAT PPDAT579={VEL 100.0,ACC 100.0,APO_DIST 100.0}
DECL E6POS XP882={x 1860.66699,y -1529.20898,z 642.863098,a 25.7857208,b -1.25422895,c 176.274002,s 2,t 34,e1 0.0,e2 0.0,e3 0.0,e4 0.0,e5 0.0,e6 0.0}
DECL FDAT FP882={TOOL_NO 1,BASE_NO 0,IPO_FRAME #BASE}
DECL PDAT PPDAT580={VEL 100.0,ACC 100.0,APO_DIST 100.0}
DECL E6POS XP883={x 1838.44995,y -1527.78796,z 608.491882,a 25.75494,b -1.242275,c 176.294006,s 2,t 34,e1 0.0,e2 0.0,e3 0.0,e4 0.0,e5 0.0,e6 0.0}
DECL FDAT FP883={TOOL_NO 1,BASE_NO 0,IPO_FRAME #BASE}
DECL LDAT LCPDAT273={VEL 2.0,ACC 100.0,APO_DIST 100.0,APO_FAC 50.0}
DECL E6POS XP884={x 1799.22998,y -1526.58801,z 608.364685,a 25.7351704,b -1.22906005,c 176.322693,s 2,t 34,e1 0.0,e2 0.0,e3 0.0,e4 0.0,e5 0.0,e6 0.0}
DECL FDAT FP884={TOOL_NO 1,BASE_NO 0,IPO_FRAME #BASE}
DECL LDAT LCPDAT274={VEL 2.0,ACC 100.0,APO_DIST 100.0,APO_FAC 50.0}
DECL E6POS XP885={x 1799.23096,y -1526.59497,z 655.081116,a 25.7347908,b -1.22934604,c 176.322205,s 2,t 34,e1 0.0,e2 0.0,e3 0.0,e4 0.0,e5 0.0,e6 0.0}
DECL FDAT FP885={TOOL_NO 1,BASE_NO 0,IPO_FRAME #BASE}
DECL LDAT LCPDAT275={VEL 2.0,ACC 100.0,APO_DIST 100.0,APO_FAC 50.0}
DECL E6POS XP886={x 1799.22803,y -1526.58496,z 719.989685,a 25.7348709,b -1.22912896,c 176.323105,s 2,t 34,e1 0.0,e2 0.0,e3 0.0,e4 0.0,e5 0.0,e6 0.0}
DECL FDAT FP886={TOOL_NO 1,BASE_NO 0,IPO_FRAME #BASE}
DECL PDAT PPDAT581={VEL 100.0,ACC 100.0,APO_DIST 100.0}
DECL E6POS XP887={x 1799.29004,y -82.3157806,z 720.017517,a 25.6821003,b -2.48299694,c 177.8004,s 2,t 34,e1 0.0,e2 0.0,e3 0.0,e4 0.0,e5 0.0,e6 0.0}
DECL FDAT FP887={TOOL_NO 1,BASE_NO 0,IPO_FRAME #BASE}
DECL PDAT PPDAT582={VEL 100.0,ACC 100.0,APO_DIST 100.0}
DECL E6POS XP888={x 1799.30701,y 860.608582,z 1382.677,a 81.5148468,b -2.00226498,c 175.8414,s 2,t 35,e1 0.0,e2 0.0,e3 0.0,e4 0.0,e5 0.0,e6 0.0}
DECL FDAT FP888={TOOL_NO 1,BASE_NO 0,IPO_FRAME #BASE}
DECL PDAT PPDAT583={VEL 100.0,ACC 100.0,APO_DIST 100.0}
DECL E6POS XP889={x 1609.86401,y 1631.90002,z 1256.89099,a 76.4038315,b -2.0085659,c 175.839798,s 2,t 35,e1 0.0,e2 0.0,e3 0.0,e4 0.0,e5 0.0,e6 0.0}
DECL FDAT FP889={TOOL_NO 1,BASE_NO 0,IPO_FRAME #BASE}
DECL PDAT PPDAT584={VEL 100.0,ACC 100.0,APO_DIST 100.0}
DECL E6POS XP890={x 1609.75696,y 1632.01196,z 1241.46594,a 76.1206207,b -2.85729408,c -178.738403,s 2,t 43,e1 0.0,e2 0.0,e3 0.0,e4 0.0,e5 0.0,e6 0.0}
DECL FDAT FP890={TOOL_NO 1,BASE_NO 0,IPO_FRAME #BASE}
DECL LDAT LCPDAT276={VEL 2.0,ACC 100.0,APO_DIST 100.0,APO_FAC 50.0}
DECL E6POS XP891={x 1609.76404,y 1634.53406,z 1227.97498,a 76.3281784,b -2.85829806,c -178.7397,s 2,t 43,e1 0.0,e2 0.0,e3 0.0,e4 0.0,e5 0.0,e6 0.0}
DECL FDAT FP891={TOOL_NO 1,BASE_NO 0,IPO_FRAME #BASE}
DECL LDAT LCPDAT277={VEL 2.0,ACC 100.0,APO_DIST 100.0,APO_FAC 50.0}
DECL E6POS XP892={x 1609.75696,y 1634.53296,z 1221.46997,a 76.3280411,b -2.85753608,c -178.739502,s 2,t 43,e1 0.0,e2 0.0,e3 0.0,e4 0.0,e5 0.0,e6 0.0}
DECL FDAT FP892={TOOL_NO 1,BASE_NO 0,IPO_FRAME #BASE}
DECL LDAT LCPDAT278={VEL 2.0,ACC 100.0,APO_DIST 100.0,APO_FAC 50.0}
DECL E6POS XP893={x 1660.14001,y 1684.52405,z 1221.47302,a 76.3276825,b -2.858459,c -178.740097,s 2,t 43,e1 0.0,e2 0.0,e3 0.0,e4 0.0,e5 0.0,e6 0.0}
DECL FDAT FP893={TOOL_NO 1,BASE_NO 0,IPO_FRAME #BASE}
DECL LDAT LCPDAT279={VEL 2.0,ACC 100.0,APO_DIST 100.0,APO_FAC 50.0}
DECL E6POS XP894={x 1660.13794,y 1684.521,z 1299.00696,a 76.3268127,b -2.858325,c -178.740097,s 2,t 43,e1 0.0,e2 0.0,e3 0.0,e4 0.0,e5 0.0,e6 0.0}
DECL FDAT FP894={TOOL_NO 1,BASE_NO 0,IPO_FRAME #BASE}
DECL PDAT PPDAT585={VEL 100.0,ACC 100.0,APO_DIST 100.0}
DECL E6POS XP895={x 1660.13794,y 1684.52197,z 1374.20496,a 76.3268738,b -2.85910106,c -178.740601,s 2,t 43,e1 0.0,e2 0.0,e3 0.0,e4 0.0,e5 0.0,e6 0.0}
DECL FDAT FP895={TOOL_NO 1,BASE_NO 0,IPO_FRAME #BASE}
DECL PDAT PPDAT586={VEL 100.0,ACC 100.0,APO_DIST 100.0}
DECL E6POS XP896={x 1675.53296,y 1393.375,z 1577.74597,a 76.3267517,b -2.85850406,c -178.740494,s 2,t 43,e1 0.0,e2 0.0,e3 0.0,e4 0.0,e5 0.0,e6 0.0}
DECL FDAT FP896={TOOL_NO 1,BASE_NO 0,IPO_FRAME #BASE}
DECL PDAT PPDAT587={VEL 100.0,ACC 100.0,APO_DIST 100.0}
DECL E6POS XP897={x 1341.71399,y -974.840027,z 988.560608,a 76.3263092,b -2.85842299,c -178.740997,s 2,t 42,e1 0.0,e2 0.0,e3 0.0,e4 0.0,e5 0.0,e6 0.0}
DECL FDAT FP897={TOOL_NO 1,BASE_NO 0,IPO_FRAME #BASE}
DECL PDAT PPDAT588={VEL 100.0,ACC 100.0,APO_DIST 100.0}
DECL E6POS XP898={x 1248.776,y -913.338989,z 845.195679,a 117.022499,b 1.62681997,c 178.727005,s 2,t 42,e1 0.0,e2 0.0,e3 0.0,e4 0.0,e5 0.0,e6 0.0}
DECL FDAT FP898={TOOL_NO 1,BASE_NO 0,IPO_FRAME #BASE}
DECL PDAT PPDAT589={VEL 100.0,ACC 100.0,APO_DIST 100.0}
DECL E6POS XP899={x 1253.00696,y -913.317383,z 598.303894,a 114.828201,b 1.62474203,c 178.729004,s 2,t 42,e1 0.0,e2 0.0,e3 0.0,e4 0.0,e5 0.0,e6 0.0}
DECL FDAT FP899={TOOL_NO 1,BASE_NO 0,IPO_FRAME #BASE}
DECL PDAT PPDAT590={VEL 100.0,ACC 100.0,APO_DIST 100.0}
DECL E6POS XP900={x 1253.01001,y -978.737122,z 592.641174,a 114.827599,b 1.62485695,c 178.728897,s 2,t 42,e1 0.0,e2 0.0,e3 0.0,e4 0.0,e5 0.0,e6 0.0}
DECL FDAT FP900={TOOL_NO 1,BASE_NO 0,IPO_FRAME #BASE}
DECL LDAT LCPDAT280={VEL 2.0,ACC 100.0,APO_DIST 100.0,APO_FAC 50.0}
DECL E6POS XP901={x 1252.77002,y -1020.51501,z 592.645874,a 114.8349,b 1.82319403,c 179.311798,s 2,t 34,e1 0.0,e2 0.0,e3 0.0,e4 0.0,e5 0.0,e6 0.0}
DECL FDAT FP901={TOOL_NO 1,BASE_NO 0,IPO_FRAME #BASE}
DECL LDAT LCPDAT281={VEL 2.0,ACC 100.0,APO_DIST 100.0,APO_FAC 50.0}
DECL E6POS XP902={x 1263.38403,y -1020.33502,z 594.706116,a 114.819801,b 2.10123897,c 178.699997,s 2,t 42,e1 0.0,e2 0.0,e3 0.0,e4 0.0,e5 0.0,e6 0.0}
DECL FDAT FP902={TOOL_NO 1,BASE_NO 0,IPO_FRAME #BASE}
DECL LDAT LCPDAT282={VEL 2.0,ACC 100.0,APO_DIST 100.0,APO_FAC 50.0}
DECL E6POS XP903={x 1263.38403,y -1020.33502,z 625.024597,a 114.819801,b 2.101403,c 178.699905,s 2,t 42,e1 0.0,e2 0.0,e3 0.0,e4 0.0,e5 0.0,e6 0.0}
DECL FDAT FP903={TOOL_NO 1,BASE_NO 0,IPO_FRAME #BASE}
DECL LDAT LCPDAT283={VEL 2.0,ACC 100.0,APO_DIST 100.0,APO_FAC 50.0}
DECL E6POS XP904={x 1263.38,y -1020.33197,z 688.816284,a 114.819298,b 2.10045004,c 178.700302,s 2,t 42,e1 0.0,e2 0.0,e3 0.0,e4 0.0,e5 0.0,e6 0.0}
DECL FDAT FP904={TOOL_NO 1,BASE_NO 0,IPO_FRAME #BASE}
DECL PDAT PPDAT591={VEL 100.0,ACC 100.0,APO_DIST 100.0}
DECL E6POS XP905={x 1263.38098,y 535.155823,z 1453.13501,a 114.819603,b 2.10045791,c 178.700195,s 2,t 35,e1 0.0,e2 0.0,e3 0.0,e4 0.0,e5 0.0,e6 0.0}
DECL FDAT FP905={TOOL_NO 1,BASE_NO 0,IPO_FRAME #BASE}
DECL PDAT PPDAT592={VEL 100.0,ACC 100.0,APO_DIST 100.0}
DECL E6POS XP906={x 897.335876,y 1571.90503,z 1453.13403,a 164.976303,b 2.10037708,c 178.700394,s 2,t 35,e1 0.0,e2 0.0,e3 0.0,e4 0.0,e5 0.0,e6 0.0}
DECL FDAT FP906={TOOL_NO 1,BASE_NO 0,IPO_FRAME #BASE}
DECL PDAT PPDAT593={VEL 100.0,ACC 100.0,APO_DIST 100.0}
DECL E6POS XP907={x 865.246094,y 1550.27197,z 1230.71497,a 166.390503,b 2.10056996,c 178.699402,s 2,t 35,e1 0.0,e2 0.0,e3 0.0,e4 0.0,e5 0.0,e6 0.0}
DECL FDAT FP907={TOOL_NO 1,BASE_NO 0,IPO_FRAME #BASE}
DECL PDAT PPDAT594={VEL 100.0,ACC 100.0,APO_DIST 100.0}
DECL E6POS XP908={x 865.25177,y 1552.198,z 1212.11304,a 166.391205,b 2.10028696,c 178.698898,s 2,t 35,e1 0.0,e2 0.0,e3 0.0,e4 0.0,e5 0.0,e6 0.0}
DECL FDAT FP908={TOOL_NO 1,BASE_NO 0,IPO_FRAME #BASE}
DECL LDAT LCPDAT284={VEL 2.0,ACC 100.0,APO_DIST 100.0,APO_FAC 50.0}
DECL E6POS XP909={x 866.094482,y 1555.01196,z 1231.22205,a 166.395401,b -0.139191896,c 176.842407,s 2,t 43,e1 0.0,e2 0.0,e3 0.0,e4 0.0,e5 0.0,e6 0.0}
DECL FDAT FP909={TOOL_NO 1,BASE_NO 0,IPO_FRAME #BASE}
DECL LDAT LCPDAT285={VEL 2.0,ACC 100.0,APO_DIST 100.0,APO_FAC 50.0}
DECL E6POS XP910={x 866.09137,y 1555.00598,z 1222.16199,a 166.395294,b -0.139310107,c 176.842804,s 2,t 43,e1 0.0,e2 0.0,e3 0.0,e4 0.0,e5 0.0,e6 0.0}
DECL FDAT FP910={TOOL_NO 1,BASE_NO 0,IPO_FRAME #BASE}
DECL LDAT LCPDAT286={VEL 2.0,ACC 100.0,APO_DIST 100.0,APO_FAC 50.0}
DECL E6POS XP911={x 809.880615,y 1554.99304,z 1222.15698,a 166.394897,b -0.139069393,c 176.843399,s 2,t 43,e1 0.0,e2 0.0,e3 0.0,e4 0.0,e5 0.0,e6 0.0}
DECL FDAT FP911={TOOL_NO 1,BASE_NO 0,IPO_FRAME #BASE}
DECL LDAT LCPDAT287={VEL 2.0,ACC 100.0,APO_DIST 100.0,APO_FAC 50.0}
DECL E6POS XP912={x 699.510376,y 1554.98901,z 1222.15002,a 166.394897,b -0.139277503,c 176.843704,s 2,t 43,e1 0.0,e2 0.0,e3 0.0,e4 0.0,e5 0.0,e6 0.0}
DECL FDAT FP912={TOOL_NO 1,BASE_NO 0,IPO_FRAME #BASE}
DECL PDAT PPDAT595={VEL 100.0,ACC 100.0,APO_DIST 100.0}
DECL E6POS XP913={x 699.511902,y 1554.98499,z 1488.83105,a 166.394501,b -0.139487296,c 176.844101,s 2,t 43,e1 0.0,e2 0.0,e3 0.0,e4 0.0,e5 0.0,e6 0.0}
DECL FDAT FP913={TOOL_NO 1,BASE_NO 0,IPO_FRAME #BASE}
DECL PDAT PPDAT596={VEL 100.0,ACC 100.0,APO_DIST 100.0}
DECL E6POS XP914={x 699.508789,y 538.287781,z 1488.85706,a 166.396896,b -0.138524607,c 176.842697,s 2,t 43,e1 0.0,e2 0.0,e3 0.0,e4 0.0,e5 0.0,e6 0.0}
DECL FDAT FP914={TOOL_NO 1,BASE_NO 0,IPO_FRAME #BASE}
DECL PDAT PPDAT597={VEL 100.0,ACC 100.0,APO_DIST 100.0}
DECL E6POS XP915={x 699.515991,y -1863.35803,z 1488.84802,a -179.705093,b -0.138834104,c 176.842194,s 2,t 10,e1 0.0,e2 0.0,e3 0.0,e4 0.0,e5 0.0,e6 0.0}
DECL FDAT FP915={TOOL_NO 1,BASE_NO 0,IPO_FRAME #BASE}
DECL PDAT PPDAT598={VEL 100.0,ACC 100.0,APO_DIST 100.0}
DECL E6POS XP916={x 1107.23206,y -2206.31201,z 732.711182,a -64.4342194,b -0.146776795,c 176.841003,s 2,t 2,e1 0.0,e2 0.0,e3 0.0,e4 0.0,e5 0.0,e6 0.0}
DECL FDAT FP916={TOOL_NO 1,BASE_NO 0,IPO_FRAME #BASE}
DECL PDAT PPDAT599={VEL 100.0,ACC 100.0,APO_DIST 100.0}
DECL E6POS XP917={x 1277.12903,y -2126.3269,z 663.030579,a -64.4268265,b -0.130556002,c 176.844498,s 2,t 2,e1 0.0,e2 0.0,e3 0.0,e4 0.0,e5 0.0,e6 0.0}
DECL FDAT FP917={TOOL_NO 1,BASE_NO 0,IPO_FRAME #BASE}
DECL PDAT PPDAT600={VEL 100.0,ACC 100.0,APO_DIST 100.0}
DECL E6POS XP918={x 1277.21802,y -2126.26196,z 611.331421,a -64.6608429,b -3.56653905,c -175.942093,s 2,t 10,e1 0.0,e2 0.0,e3 0.0,e4 0.0,e5 0.0,e6 0.0}
DECL FDAT FP918={TOOL_NO 1,BASE_NO 0,IPO_FRAME #BASE}
DECL PDAT PPDAT601={VEL 100.0,ACC 100.0,APO_DIST 100.0}
DECL E6POS XP919={x 1276.80005,y -2112.41504,z 611.11322,a -64.6627884,b -3.54889011,c -175.948807,s 2,t 10,e1 0.0,e2 0.0,e3 0.0,e4 0.0,e5 0.0,e6 0.0}
DECL FDAT FP919={TOOL_NO 1,BASE_NO 0,IPO_FRAME #BASE}
DECL LDAT LCPDAT288={VEL 2.0,ACC 100.0,APO_DIST 100.0,APO_FAC 50.0}
DECL E6POS XP920={x 1276.58801,y -2080.27588,z 611.015381,a -64.6592026,b -3.53906202,c -175.953995,s 2,t 10,e1 0.0,e2 0.0,e3 0.0,e4 0.0,e5 0.0,e6 0.0}
DECL FDAT FP920={TOOL_NO 1,BASE_NO 0,IPO_FRAME #BASE}
DECL LDAT LCPDAT289={VEL 2.0,ACC 100.0,APO_DIST 100.0,APO_FAC 50.0}
DECL E6POS XP921={x 1276.58801,y -2080.28003,z 671.877808,a -64.6594162,b -3.53952503,c -175.954407,s 2,t 10,e1 0.0,e2 0.0,e3 0.0,e4 0.0,e5 0.0,e6 0.0}
DECL FDAT FP921={TOOL_NO 1,BASE_NO 0,IPO_FRAME #BASE}
DECL LDAT LCPDAT290={VEL 2.0,ACC 100.0,APO_DIST 100.0,APO_FAC 50.0}
DECL E6POS XP922={x 1276.58704,y -2080.28296,z 777.328674,a -64.6594772,b -3.53981996,c -175.954697,s 2,t 10,e1 0.0,e2 0.0,e3 0.0,e4 0.0,e5 0.0,e6 0.0}
DECL FDAT FP922={TOOL_NO 1,BASE_NO 0,IPO_FRAME #BASE}
DECL PDAT PPDAT602={VEL 100.0,ACC 100.0,APO_DIST 100.0}
DECL E6POS XP923={x 1276.58801,y -2080.28394,z 1232.85303,a -64.6595078,b -3.54048896,c -175.954605,s 2,t 10,e1 0.0,e2 0.0,e3 0.0,e4 0.0,e5 0.0,e6 0.0}
DECL FDAT FP923={TOOL_NO 1,BASE_NO 0,IPO_FRAME #BASE}
DECL PDAT PPDAT603={VEL 100.0,ACC 100.0,APO_DIST 100.0}
DECL E6POS XP924={x 1276.58606,y 455.985413,z 1340.87097,a -64.7281418,b 1.18211102,c -173.376801,s 2,t 11,e1 0.0,e2 0.0,e3 0.0,e4 0.0,e5 0.0,e6 0.0}
DECL FDAT FP924={TOOL_NO 1,BASE_NO 0,IPO_FRAME #BASE}
DECL PDAT PPDAT604={VEL 100.0,ACC 100.0,APO_DIST 100.0}
DECL E6POS XP925={x 1740.078,y 702.766418,z 1340.85303,a -4.79579878,b 1.18323004,c -173.377304,s 2,t 11,e1 0.0,e2 0.0,e3 0.0,e4 0.0,e5 0.0,e6 0.0}
DECL FDAT FP925={TOOL_NO 1,BASE_NO 0,IPO_FRAME #BASE}
DECL PDAT PPDAT605={VEL 100.0,ACC 100.0,APO_DIST 100.0}
DECL E6POS XP926={x 1710.87805,y 890.413818,z 1240.81897,a -13.7459402,b -1.86556697,c -172.673004,s 2,t 11,e1 0.0,e2 0.0,e3 0.0,e4 0.0,e5 0.0,e6 0.0}
DECL FDAT FP926={TOOL_NO 1,BASE_NO 0,IPO_FRAME #BASE}
DECL LDAT LCPDAT291={VEL 2.0,ACC 100.0,APO_DIST 100.0,APO_FAC 50.0}
DECL E6POS XP927={x 1710.86304,y 892.215027,z 1241.10303,a -13.7396097,b -0.477629811,c -173.013107,s 2,t 11,e1 0.0,e2 0.0,e3 0.0,e4 0.0,e5 0.0,e6 0.0}
DECL FDAT FP927={TOOL_NO 1,BASE_NO 0,IPO_FRAME #BASE}
DECL LDAT LCPDAT292={VEL 2.0,ACC 100.0,APO_DIST 100.0,APO_FAC 50.0}
DECL E6POS XP928={x 1710.86804,y 892.217712,z 1218.80005,a -13.7402,b -0.477732599,c -173.012894,s 2,t 11,e1 0.0,e2 0.0,e3 0.0,e4 0.0,e5 0.0,e6 0.0}
DECL FDAT FP928={TOOL_NO 1,BASE_NO 0,IPO_FRAME #BASE}
DECL LDAT LCPDAT293={VEL 2.0,ACC 100.0,APO_DIST 100.0,APO_FAC 50.0}
DECL E6POS XP929={x 1756.76794,y 863.957092,z 1218.83301,a -13.7429399,b -0.478674293,c -173.011002,s 2,t 11,e1 0.0,e2 0.0,e3 0.0,e4 0.0,e5 0.0,e6 0.0}
DECL FDAT FP929={TOOL_NO 1,BASE_NO 0,IPO_FRAME #BASE}
DECL LDAT LCPDAT294={VEL 2.0,ACC 100.0,APO_DIST 100.0,APO_FAC 50.0}
DECL E6POS XP930={x 1756.78601,y 581.483887,z 1389.80603,a -13.7413702,b -0.481534809,c -173.010101,s 2,t 11,e1 0.0,e2 0.0,e3 0.0,e4 0.0,e5 0.0,e6 0.0}
DECL FDAT FP930={TOOL_NO 1,BASE_NO 0,IPO_FRAME #BASE}
DECL PDAT PPDAT606={VEL 100.0,ACC 100.0,APO_DIST 100.0}
DECL E6POS XP931={x -2509.7251,y 974.890686,z 1358.58997,a -21.2311897,b 84.7598572,c 179.997192,s 2,t 35,e1 0.0,e2 0.0,e3 0.0,e4 0.0,e5 0.0,e6 0.0}
DECL FDAT FP931={TOOL_NO 1,BASE_NO 0,IPO_FRAME #BASE}
DECL PDAT PPDAT607={VEL 100.0,ACC 100.0,APO_DIST 100.0}
DECL E6POS XP932={x -13.3743801,y 417.108002,z 2611.2251,a 91.8369064,b -6.43569803,c -4.21044206E-05,s 0,t 39,e1 0.0,e2 0.0,e3 0.0,e4 0.0,e5 0.0,e6 0.0}
DECL FDAT FP932={TOOL_NO 1,BASE_NO 0,IPO_FRAME #BASE}
DECL PDAT PPDAT608={VEL 100.0,ACC 100.0,APO_DIST 100.0}
DECL E6POS XP933={x -13.3708296,y 416.967285,z 3257.58594,a 91.8382416,b -6.45274115,c -0.000194934299,s 4,t 55,e1 0.0,e2 0.0,e3 0.0,e4 0.0,e5 0.0,e6 0.0}
DECL FDAT FP933={TOOL_NO 1,BASE_NO 0,IPO_FRAME #BASE}
DECL PDAT PPDAT609={VEL 100.0,ACC 100.0,APO_DIST 100.0}
DECL E6POS XP934={x -10.2149401,y 318.550903,z 3250.76099,a 91.8382416,b -2.92804408,c -9.71544723E-05,s 6,t 51,e1 0.0,e2 0.0,e3 0.0,e4 0.0,e5 0.0,e6 0.0}
DECL FDAT FP934={TOOL_NO 1,BASE_NO 0,IPO_FRAME #BASE}
DECL PDAT PPDAT610={VEL 100.0,ACC 100.0,APO_DIST 100.0}
DECL E6POS XP935={x -10.2165699,y 318.544312,z 2793.10303,a 91.8378601,b -2.93255401,c -0.000167870196,s 6,t 51,e1 0.0,e2 0.0,e3 0.0,e4 0.0,e5 0.0,e6 0.0}
DECL FDAT FP935={TOOL_NO 1,BASE_NO 0,IPO_FRAME #BASE}
DECL PDAT PPDAT611={VEL 100.0,ACC 100.0,APO_DIST 100.0}
DECL E6POS XP936={x -10.2218103,y 583.397705,z 1915.35498,a 91.8411179,b -2.93410707,c -0.000434148009,s 6,t 59,e1 0.0,e2 0.0,e3 0.0,e4 0.0,e5 0.0,e6 0.0}
DECL FDAT FP936={TOOL_NO 1,BASE_NO 0,IPO_FRAME #BASE}
DECL PDAT PPDAT612={VEL 100.0,ACC 100.0,APO_DIST 100.0}
DECL E6POS XP937={x -15.3889599,y 866.633423,z 1662.76794,a 104.634201,b 86.2745667,c 13.6017399,s 6,t 59,e1 0.0,e2 0.0,e3 0.0,e4 0.0,e5 0.0,e6 0.0}
DECL FDAT FP937={TOOL_NO 1,BASE_NO 0,IPO_FRAME #BASE}
DECL PDAT PPDAT613={VEL 100.0,ACC 100.0,APO_DIST 100.0}
DECL E6POS XP938={x -15.50881,y 2620.979,z 1663.44897,a 103.9627,b 86.2529221,c 12.9073296,s 6,t 51,e1 0.0,e2 0.0,e3 0.0,e4 0.0,e5 0.0,e6 0.0}
DECL FDAT FP938={TOOL_NO 1,BASE_NO 0,IPO_FRAME #BASE}
DECL PDAT PPDAT614={VEL 100.0,ACC 100.0,APO_DIST 100.0}
DECL E6POS XP939={x -1611.81702,y -50.8759003,z 1663.43896,a -164.780807,b 86.2533264,c 12.90732,s 6,t 51,e1 0.0,e2 0.0,e3 0.0,e4 0.0,e5 0.0,e6 0.0}
DECL FDAT FP939={TOOL_NO 1,BASE_NO 0,IPO_FRAME #BASE}
DECL PDAT PPDAT615={VEL 100.0,ACC 100.0,APO_DIST 100.0}
DECL E6POS XP940={x -2088.22607,y -50.879631,z 1663.45105,a -164.782394,b 86.2527924,c 12.90553,s 6,t 51,e1 0.0,e2 0.0,e3 0.0,e4 0.0,e5 0.0,e6 0.0}
DECL FDAT FP940={TOOL_NO 1,BASE_NO 0,IPO_FRAME #BASE}
DECL PDAT PPDAT616={VEL 100.0,ACC 100.0,APO_DIST 100.0}
DECL E6POS XP941={x -2738.05005,y -50.9311981,z 1357.505,a -164.778397,b 86.2501373,c 12.9014702,s 6,t 51,e1 0.0,e2 0.0,e3 0.0,e4 0.0,e5 0.0,e6 0.0}
DECL FDAT FP941={TOOL_NO 1,BASE_NO 0,IPO_FRAME #BASE}
DECL PDAT PPDAT617={VEL 100.0,ACC 100.0,APO_DIST 100.0}
DECL E6POS XP942={x -2725.33691,y -50.8927002,z 1357.13696,a -164.467697,b 86.2582779,c 13.21696,s 6,t 51,e1 0.0,e2 0.0,e3 0.0,e4 0.0,e5 0.0,e6 0.0}
DECL FDAT FP942={TOOL_NO 1,BASE_NO 0,IPO_FRAME #BASE}
DECL PDAT PPDAT618={VEL 100.0,ACC 100.0,APO_DIST 100.0}
DECL E6POS XP943={x -943.853088,y -558.490173,z 2387.33496,a 62.3781815,b 37.3523216,c -159.4104,s 2,t 2,e1 0.0,e2 0.0,e3 0.0,e4 0.0,e5 0.0,e6 0.0}
DECL FDAT FP943={TOOL_NO 1,BASE_NO 0,IPO_FRAME #BASE}
DECL PDAT PPDAT619={VEL 100.0,ACC 100.0,APO_DIST 100.0}
DECL E6POS XP944={x -1316.61902,y -574.356201,z 2652.31299,a -174.126694,b -0.464748204,c 0.213377103,s 6,t 26,e1 0.0,e2 0.0,e3 0.0,e4 0.0,e5 0.0,e6 0.0}
DECL FDAT FP944={TOOL_NO 1,BASE_NO 0,IPO_FRAME #BASE}
DECL PDAT PPDAT620={VEL 100.0,ACC 100.0,APO_DIST 100.0}
DECL E6POS XP945={x -1210.203,y -573.858521,z 3072.52808,a -174.103897,b -0.473572791,c 0.216105893,s 6,t 26,e1 0.0,e2 0.0,e3 0.0,e4 0.0,e5 0.0,e6 0.0}
DECL FDAT FP945={TOOL_NO 1,BASE_NO 0,IPO_FRAME #BASE}
DECL PDAT PPDAT621={VEL 100.0,ACC 100.0,APO_DIST 100.0}
DECL E6POS XP946={x -1210.198,y -573.852722,z 2853.54907,a -174.106201,b -0.470291287,c 0.215059996,s 6,t 26,e1 0.0,e2 0.0,e3 0.0,e4 0.0,e5 0.0,e6 0.0}
DECL FDAT FP946={TOOL_NO 1,BASE_NO 0,IPO_FRAME #BASE}
DECL PDAT PPDAT622={VEL 100.0,ACC 100.0,APO_DIST 100.0}
DECL E6POS XP947={x 1091.66003,y -905.758972,z 2070.11011,a -174.107101,b -0.470405102,c 0.215554997,s 6,t 18,e1 0.0,e2 0.0,e3 0.0,e4 0.0,e5 0.0,e6 0.0}
DECL FDAT FP947={TOOL_NO 1,BASE_NO 0,IPO_FRAME #BASE}
DECL PDAT PPDAT623={VEL 100.0,ACC 100.0,APO_DIST 100.0}
DECL E6POS XP948={x 2120.80688,y 3.5303719,z 1206.47998,a -9.48567009,b 87.1038437,c -9.64396763,s 6,t 19,e1 0.0,e2 0.0,e3 0.0,e4 0.0,e5 0.0,e6 0.0}
DECL FDAT FP948={TOOL_NO 1,BASE_NO 0,IPO_FRAME #BASE}
DECL PDAT PPDAT624={VEL 100.0,ACC 100.0,APO_DIST 100.0}
DECL E6POS XP949={x 1619.87305,y -0.00344022503,z 2797.35693,a 7.16774607,b 89.9810867,c 7.16786718,s 2,t 34,e1 0.0,e2 0.0,e3 0.0,e4 0.0,e5 0.0,e6 0.0}
DECL FDAT FP949={TOOL_NO 1,BASE_NO 0,IPO_FRAME #BASE}
DECL PDAT PPDAT625={VEL 100.0,ACC 100.0,APO_DIST 100.0}
DECL E6POS XP950={x 549.078613,y 362.529114,z 2742.34204,a -50.0954514,b 89.8847275,c -50.0885391,s 3,t 42,e1 0.0,e2 0.0,e3 0.0,e4 0.0,e5 0.0,e6 0.0}
DECL FDAT FP950={TOOL_NO 1,BASE_NO 0,IPO_FRAME #BASE}
DECL PDAT PPDAT626={VEL 100.0,ACC 100.0,APO_DIST 100.0}
DECL E6POS XP951={x 597.747314,y -516.802979,z 1744.46802,a -88.9560165,b -26.5237904,c -86.5755234,s 6,t 18,e1 0.0,e2 0.0,e3 0.0,e4 0.0,e5 0.0,e6 0.0}
DECL FDAT FP951={TOOL_NO 1,BASE_NO 0,IPO_FRAME #BASE}
DECL PDAT PPDAT627={VEL 100.0,ACC 100.0,APO_DIST 100.0}
DECL E6POS XP952={x -1619.99805,y 5.61712885,z 2195.02197,a 130.729095,b 89.9915619,c -49.0722313,s 6,t 18,e1 0.0,e2 0.0,e3 0.0,e4 0.0,e5 0.0,e6 0.0}
DECL FDAT FP952={TOOL_NO 1,BASE_NO 0,IPO_FRAME #BASE}
DECL PDAT PPDAT628={VEL 100.0,ACC 100.0,APO_DIST 100.0}
DECL E6POS XP953={x -21.5673199,y 1619.86401,z 2195.03198,a 43.3751984,b 89.9911194,c -47.3875999,s 6,t 19,e1 0.0,e2 0.0,e3 0.0,e4 0.0,e5 0.0,e6 0.0}
DECL FDAT FP953={TOOL_NO 1,BASE_NO 0,IPO_FRAME #BASE}
DECL PDAT PPDAT629={VEL 100.0,ACC 100.0,APO_DIST 100.0}
DECL E6POS XP954={x -1619.99304,y 7.45334482,z 2195.03003,a 130.686096,b 89.9910126,c -49.0503197,s 6,t 19,e1 0.0,e2 0.0,e3 0.0,e4 0.0,e5 0.0,e6 0.0}
DECL FDAT FP954={TOOL_NO 1,BASE_NO 0,IPO_FRAME #BASE}
DECL PDAT PPDAT630={VEL 100.0,ACC 100.0,APO_DIST 100.0}
DECL E6POS XP955={x 1620.00305,y 4.55179596,z 2195.03491,a -47.6838608,b 89.9906235,c -47.844841,s 6,t 19,e1 0.0,e2 0.0,e3 0.0,e4 0.0,e5 0.0,e6 0.0}
DECL FDAT FP955={TOOL_NO 1,BASE_NO 0,IPO_FRAME #BASE}
DECL PDAT PPDAT631={VEL 100.0,ACC 100.0,APO_DIST 100.0}
DECL E6POS XP956={x 2136.29004,y 5.99789286,z 1160.48096,a -179.828705,b 48.8600502,c -179.992096,s 6,t 19,e1 0.0,e2 0.0,e3 0.0,e4 0.0,e5 0.0,e6 0.0}
DECL FDAT FP956={TOOL_NO 1,BASE_NO 0,IPO_FRAME #BASE}
DECL PDAT PPDAT632={VEL 100.0,ACC 100.0,APO_DIST 100.0}
DECL E6POS XP957={x 641.488525,y 1.79969394,z 2629.06396,a 0.149445593,b 52.0217094,c -0.00890493207,s 6,t 19,e1 0.0,e2 0.0,e3 0.0,e4 0.0,e5 0.0,e6 0.0}
DECL FDAT FP957={TOOL_NO 1,BASE_NO 0,IPO_FRAME #BASE}
DECL PDAT PPDAT633={VEL 100.0,ACC 100.0,APO_DIST 100.0}
DECL E6POS XP958={x 1579.96704,y 4.43259287,z 2231.05591,a -0.0509101115,b 88.1177521,c -0.211538702,s 6,t 19,e1 0.0,e2 0.0,e3 0.0,e4 0.0,e5 0.0,e6 0.0}
DECL FDAT FP958={TOOL_NO 1,BASE_NO 0,IPO_FRAME #BASE}
DECL PDAT PPDAT634={VEL 100.0,ACC 100.0,APO_DIST 100.0}
DECL E6POS XP959={x 1064.24304,y 2.98573089,z 1193.24695,a -179.830994,b 29.6551304,c -179.995895,s 6,t 19,e1 0.0,e2 0.0,e3 0.0,e4 0.0,e5 0.0,e6 0.0}
DECL FDAT FP959={TOOL_NO 1,BASE_NO 0,IPO_FRAME #BASE}
DECL PDAT PPDAT635={VEL 100.0,ACC 100.0,APO_DIST 100.0}
DECL E6POS XP960={x 354.107788,y 0.993448615,z 3255.49707,a 0.153528303,b -2.73342395,c 0.000344017812,s 4,t 23,e1 0.0,e2 0.0,e3 0.0,e4 0.0,e5 0.0,e6 0.0}
DECL FDAT FP960={TOOL_NO 1,BASE_NO 0,IPO_FRAME #BASE}
DECL PDAT PPDAT636={VEL 100.0,ACC 100.0,APO_DIST 100.0}
DECL E6POS XP961={x -651.770996,y -1.82715702,z 2012.45801,a -179.727493,b -86.3076096,c 179.888306,s 5,t 23,e1 0.0,e2 0.0,e3 0.0,e4 0.0,e5 0.0,e6 0.0}
DECL FDAT FP961={TOOL_NO 1,BASE_NO 0,IPO_FRAME #BASE}
DECL PDAT PPDAT637={VEL 100.0,ACC 100.0,APO_DIST 100.0}
DECL E6POS XP962={x 355.359497,y 0.995450616,z 3255.61792,a 0.153285295,b -2.66917491,c 0.000335919089,s 4,t 23,e1 0.0,e2 0.0,e3 0.0,e4 0.0,e5 0.0,e6 0.0}
DECL FDAT FP962={TOOL_NO 1,BASE_NO 0,IPO_FRAME #BASE}
DECL PDAT PPDAT638={VEL 100.0,ACC 100.0,APO_DIST 100.0}
DECL E6POS XP963={x 1577.27405,y 4.41498804,z 2259.40698,a 0.0365776718,b 86.6623535,c -0.12359,s 6,t 19,e1 0.0,e2 0.0,e3 0.0,e4 0.0,e5 0.0,e6 0.0}
DECL FDAT FP963={TOOL_NO 1,BASE_NO 0,IPO_FRAME #BASE}
DECL PDAT PPDAT639={VEL 100.0,ACC 100.0,APO_DIST 100.0}
DECL E6POS XP964={x 1577.276,y 4.4170661,z 2259.35693,a -130.744904,b -84.9290771,c -48.9830093,s 6,t 19,e1 0.0,e2 0.0,e3 0.0,e4 0.0,e5 0.0,e6 0.0}
DECL FDAT FP964={TOOL_NO 1,BASE_NO 0,IPO_FRAME #BASE}
DECL PDAT PPDAT640={VEL 100.0,ACC 100.0,APO_DIST 100.0}
DECL E6POS XP965={x 1577.27197,y 4.40356779,z 2259.42407,a 81.8434067,b 68.0312424,c 81.044632,s 6,t 19,e1 0.0,e2 0.0,e3 0.0,e4 0.0,e5 0.0,e6 0.0}
DECL FDAT FP965={TOOL_NO 1,BASE_NO 0,IPO_FRAME #BASE}
DECL PDAT PPDAT641={VEL 100.0,ACC 100.0,APO_DIST 100.0}
DECL E6POS XP966={x 1577.271,y 4.41558218,z 2259.43506,a -18.8469009,b 86.4686127,c -18.9738903,s 6,t 19,e1 0.0,e2 0.0,e3 0.0,e4 0.0,e5 0.0,e6 0.0}
DECL FDAT FP966={TOOL_NO 1,BASE_NO 0,IPO_FRAME #BASE}
DECL PDAT PPDAT642={VEL 100.0,ACC 100.0,APO_DIST 100.0}
DECL E6POS XP967={x 1577.27002,y 4.42778587,z 2259.44702,a -81.9723816,b 66.9015198,c -81.4597626,s 6,t 27,e1 0.0,e2 0.0,e3 0.0,e4 0.0,e5 0.0,e6 0.0}
DECL FDAT FP967={TOOL_NO 1,BASE_NO 0,IPO_FRAME #BASE}
DECL PDAT PPDAT643={VEL 100.0,ACC 100.0,APO_DIST 100.0}
DECL E6POS XP968={x 1577.26904,y 4.41508913,z 2259.45898,a -3.36278796,b 86.6526184,c -3.51719403,s 6,t 19,e1 0.0,e2 0.0,e3 0.0,e4 0.0,e5 0.0,e6 0.0}
DECL FDAT FP968={TOOL_NO 1,BASE_NO 0,IPO_FRAME #BASE}
DECL PDAT PPDAT644={VEL 100.0,ACC 100.0,APO_DIST 100.0}
DECL E6POS XP969={x 1203.97095,y 2.52681994,z 1994.46704,a -179.926895,b -22.6002808,c -179.787506,s 2,t 3,e1 0.0,e2 0.0,e3 0.0,e4 0.0,e5 0.0,e6 0.0}
DECL FDAT FP969={TOOL_NO 1,BASE_NO 0,IPO_FRAME #BASE}
DECL PDAT PPDAT645={VEL 100.0,ACC 100.0,APO_DIST 100.0}
DECL E6POS XP970={x 1577.56201,y 4.32842016,z 2234.25488,a -174.033997,b 87.9775772,c -174.179504,s 2,t 3,e1 0.0,e2 0.0,e3 0.0,e4 0.0,e5 0.0,e6 0.0}
DECL FDAT FP970={TOOL_NO 1,BASE_NO 0,IPO_FRAME #BASE}
DECL PDAT PPDAT646={VEL 100.0,ACC 100.0,APO_DIST 100.0}
DECL E6POS XP971={x 1576.52905,y 4.44661093,z 2269.14893,a -2.0193119,b 84.597229,c -2.17716789,s 6,t 19,e1 0.0,e2 0.0,e3 0.0,e4 0.0,e5 0.0,e6 0.0}
DECL FDAT FP971={TOOL_NO 1,BASE_NO 0,IPO_FRAME #BASE}
DECL PDAT PPDAT647={VEL 100.0,ACC 100.0,APO_DIST 100.0}
DECL E6POS XP972={x 1576.52698,y 4.44325876,z 2269.1709,a 82.3295364,b 55.2709808,c 80.4915009,s 6,t 19,e1 0.0,e2 0.0,e3 0.0,e4 0.0,e5 0.0,e6 0.0}
DECL FDAT FP972={TOOL_NO 1,BASE_NO 0,IPO_FRAME #BASE}
DECL PDAT PPDAT648={VEL 100.0,ACC 100.0,APO_DIST 100.0}
DECL E6POS XP973={x 1576.526,y 4.44657803,z 2269.17798,a -78.2994003,b 64.6933517,c -77.2806931,s 6,t 51,e1 0.0,e2 0.0,e3 0.0,e4 0.0,e5 0.0,e6 0.0}
DECL FDAT FP973={TOOL_NO 1,BASE_NO 0,IPO_FRAME #BASE}
DECL PDAT PPDAT649={VEL 100.0,ACC 100.0,APO_DIST 100.0}
DECL E6POS XP974={x 1576.52295,y 4.44319201,z 2269.18799,a -10.3022699,b 84.5081482,c -10.4226999,s 6,t 19,e1 0.0,e2 0.0,e3 0.0,e4 0.0,e5 0.0,e6 0.0}
DECL FDAT FP974={TOOL_NO 1,BASE_NO 0,IPO_FRAME #BASE}
DECL PDAT PPDAT650={VEL 100.0,ACC 100.0,APO_DIST 100.0}
ENDDAT
